# EPICS alarm handler configuration: mps_database/bare/alarms/areas/mpln_undh_mp01.alhConfig
GROUP NULL MPLN:UNDH:MP01:1
$ALIAS MPS Link Node 136
$GUIDANCE
LTUH MPS
   Group Name: MPLN:UNDH:MP01:1
   Summary PV:  MPLN:UNDH:MP01:1:STATSUMY
$END
CHANNEL  MPLN:UNDH:MP01:1    MPLN:UNDH:MP01:1:MPS_EN_RBV		-----
CHANNEL  MPLN:UNDH:MP01:1    MPLN:UNDH:MP01:1:LC1_MODE_RBV		-----
